(* Logix 5000 project; controller Amvex_Thorpe_Flowmeter vendor 1 type 14 code 106 rev 33.13; software revision 33.01; part 12 of 16 *)
(* tags used below, declared in another part *)
   Auto_Seq : SEQ;
   Barcode_Latch : BOOL;
   Barcode_Result_DATA : SINT[128];
   FAULTED : DINT;
   InfeedPalletTM1 : TIMER;
   Lift_stop_timer : TIMER;
   Manual_ONS : BOOL;
   MODE : MODE;
   Part_count : DINT;
   Test : Connect;
   Test_ONS : BOOL[32];
   Barcode_Data_String : STRING;
   Barcode_Delay : TIMER;
   Close : BOOL;
   Close_Rapid : Servo_Move;
   Close_Step : Servo_Move;
   Empty_Pallet_Timer : TIMER;
   Empty_Pallet_Timer2 : TIMER;
   Fastest_Delay : TIMER;
   In_Cycle : BOOL;
   Last_Test_Data : REAL[8];
   MCP : MCP;
   Open : BOOL;
   PH_Debug : DINT;
   Reject : BOOL;
   Reject_Barcode : BOOL;
   Reject_Pallet_Bit : DINT;
   Safety_OK : BOOL;
   Test2_Step : Servo_Move;
   Test3_Step : Servo_Move;
   Test4_Step : Servo_Move;
   Test5_Step : Servo_Move;
   Test_Data : REAL[8];
   Test_Data_Moved : BOOL;
   Test_Data_ONS : BOOL[32];
   Test_Delay_TMR : TIMER[5];
   Transmit_Data : BOOL;
   Vision_Result_OK_TMR : TIMER[6];
   Vision_TMR : TIMER[3];
(* MCP_Main, continued *)

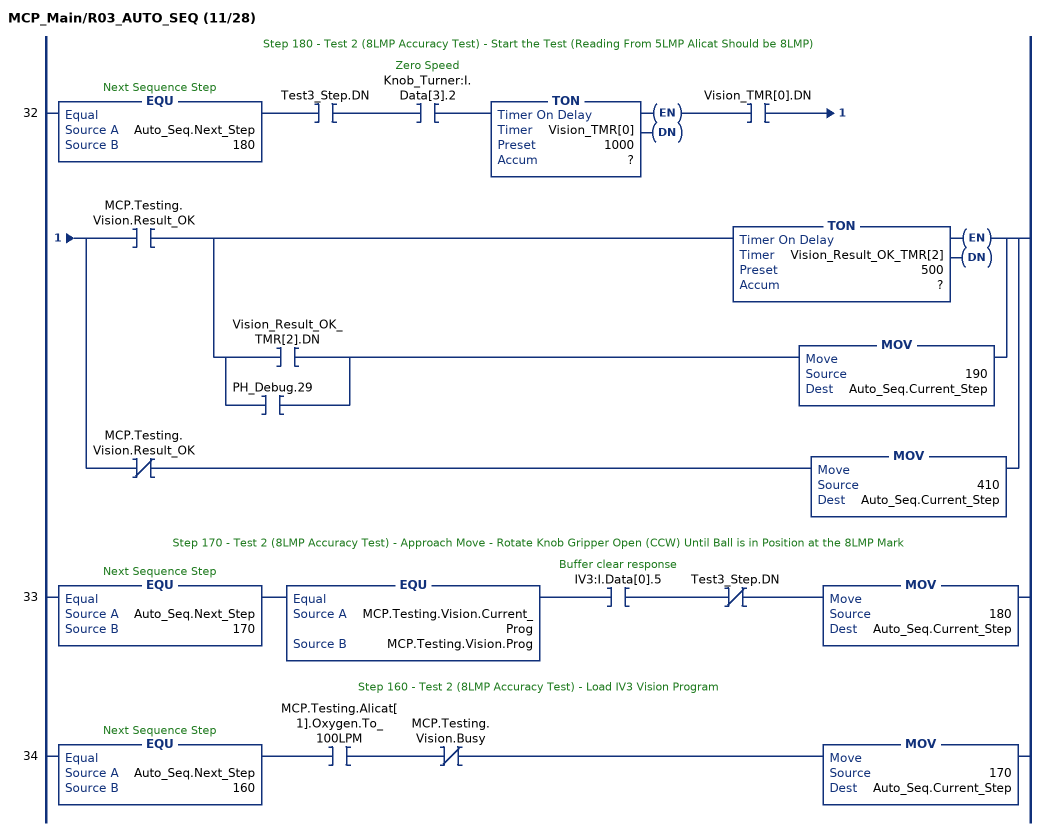
   [picture p212: MCP_Main/R03_AUTO_SEQ rungs 32-34]
   // Step 180 - Test 2 (8LMP Accuracy Test) - Start the Test (Reading From 5LMP Alicat Should be 8LMP)
   32: EQU(Auto_Seq.Next_Step,180)XIC(Test3_Step.DN)XIC(Knob_Turner:I.Data[3].2)TON(Vision_TMR[0],?,?)XIC(Vision_TMR[0].DN)[XIC(MCP.Testing.Vision.Result_OK) [TON(Vision_Result_OK_TMR[2],?,?) ,[XIC(Vision_Result_OK_TMR[2].DN) ,XIC(PH_Debug.29) ] MOV(190,Auto_Seq.Current_Step) ] ,XIO(MCP.Testing.Vision.Result_OK) MOV(410,Auto_Seq.Current_Step) ];
   // Step 170 - Test 2 (8LMP Accuracy Test) - Approach Move - Rotate Knob Gripper Open (CCW) Until Ball is in Position at the 8LMP Mark
   33: EQU(Auto_Seq.Next_Step,170)EQU(MCP.Testing.Vision.Current_Prog,MCP.Testing.Vision.Prog)XIC(IV3:I.Data[0].5)XIO(Test3_Step.DN)MOV(180,Auto_Seq.Current_Step);
   // Step 160 - Test 2 (8LMP Accuracy Test) - Load IV3 Vision Program
   34: EQU(Auto_Seq.Next_Step,160)XIC(MCP.Testing.Alicat[1].Oxygen.To_100LPM)XIO(MCP.Testing.Vision.Busy)MOV(170,Auto_Seq.Current_Step);
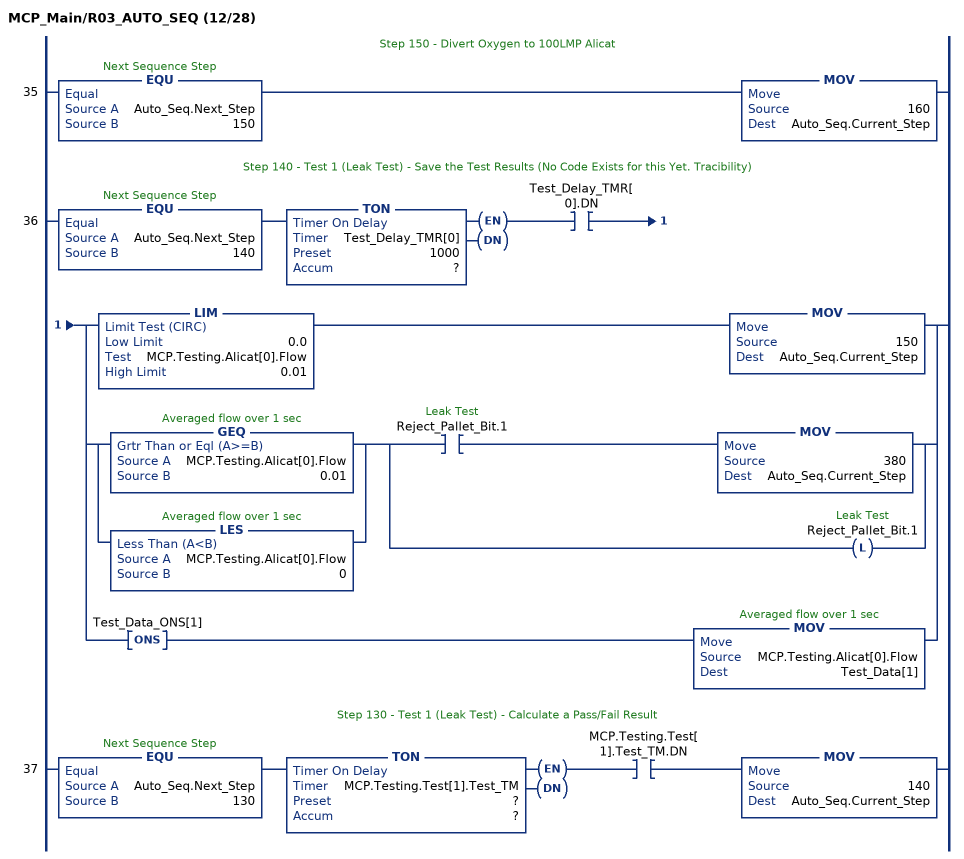
   // Step 150 - Divert Oxygen to 100LMP Alicat
   35: EQU(Auto_Seq.Next_Step,150)MOV(160,Auto_Seq.Current_Step);
   // Step 140 - Test 1 (Leak Test) - Save the Test Results (No Code Exists for this Yet. Tracibility)
   36: EQU(Auto_Seq.Next_Step,140)TON(Test_Delay_TMR[0],?,?)XIC(Test_Delay_TMR[0].DN)[LIM(0.0,MCP.Testing.Alicat[0].Flow,0.01) MOV(150,Auto_Seq.Current_Step) ,[GEQ(MCP.Testing.Alicat[0].Flow,0.01) ,LES(MCP.Testing.Alicat[0].Flow,0) ] [XIC(Reject_Pallet_Bit.1) MOV(380,Auto_Seq.Current_Step) ,OTL(Reject_Pallet_Bit.1) ] ,ONS(Test_Data_ONS[1]) MOV(MCP.Testing.Alicat[0].Flow,Test_Data[1]) ];
   // Step 130 - Test 1 (Leak Test) - Calculate a Pass/Fail Result
   37: EQU(Auto_Seq.Next_Step,130)TON(MCP.Testing.Test[1].Test_TM,?,?)XIC(MCP.Testing.Test[1].Test_TM.DN)MOV(140,Auto_Seq.Current_Step);
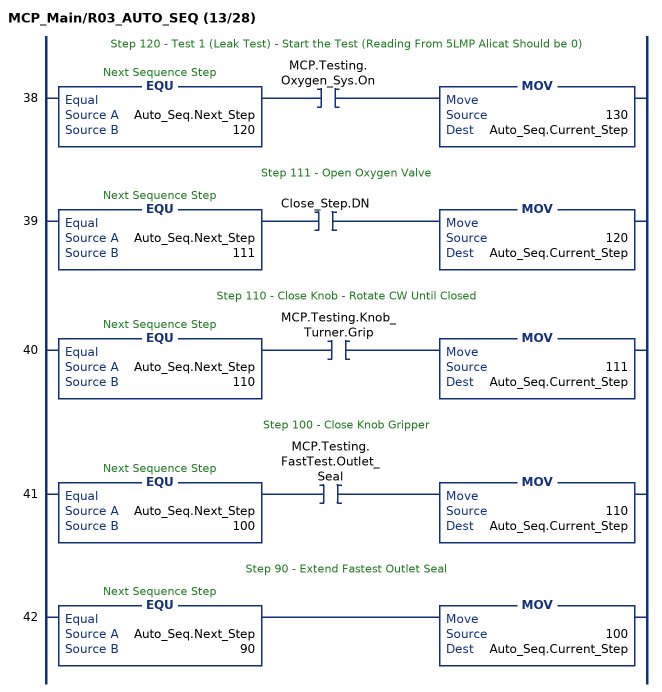
   // Step 120 - Test 1 (Leak Test) - Start the Test (Reading From 5LMP Alicat Should be 0)
   38: EQU(Auto_Seq.Next_Step,120)XIC(MCP.Testing.Oxygen_Sys.On)MOV(130,Auto_Seq.Current_Step);
   // Step 111 - Open Oxygen Valve
   39: EQU(Auto_Seq.Next_Step,111)XIC(Close_Step.DN)MOV(120,Auto_Seq.Current_Step);
   // Step 110 - Close Knob - Rotate CW Until Closed
   40: EQU(Auto_Seq.Next_Step,110)XIC(MCP.Testing.Knob_Turner.Grip)MOV(111,Auto_Seq.Current_Step);
   // Step 100 - Close Knob Gripper
   41: EQU(Auto_Seq.Next_Step,100)XIC(MCP.Testing.FastTest.Outlet_Seal)MOV(110,Auto_Seq.Current_Step);
   // Step 90 - Extend Fastest Outlet Seal
   42: EQU(Auto_Seq.Next_Step,90)MOV(100,Auto_Seq.Current_Step);
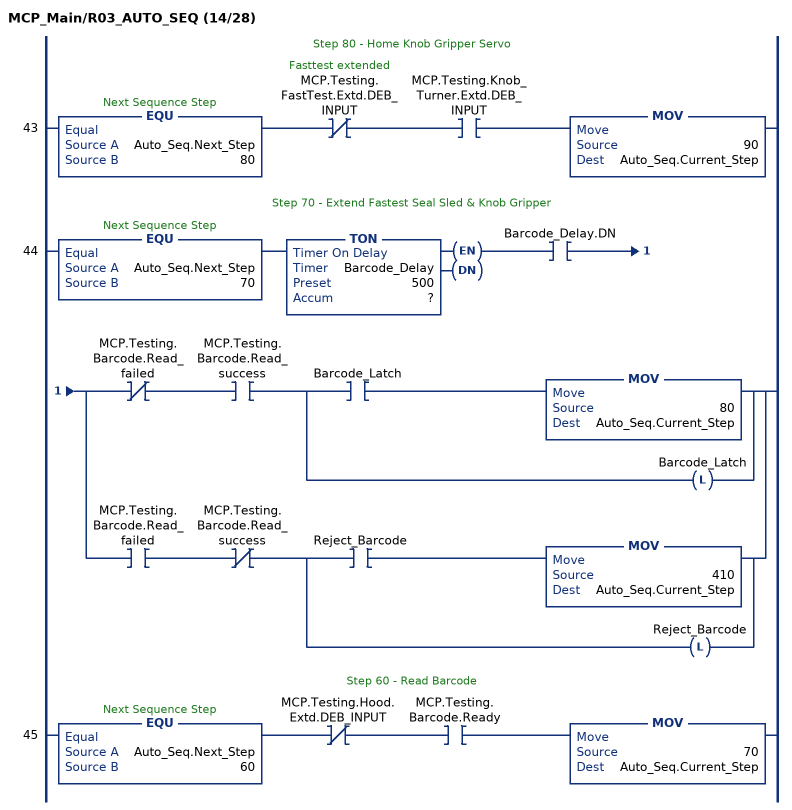
   // Step 80 - Home Knob Gripper Servo
   43: EQU(Auto_Seq.Next_Step,80)XIO(MCP.Testing.FastTest.Extd.DEB_INPUT)XIC(MCP.Testing.Knob_Turner.Extd.DEB_INPUT)MOV(90,Auto_Seq.Current_Step);
   // Step 70 - Extend Fastest Seal Sled & Knob Gripper
   44: EQU(Auto_Seq.Next_Step,70)TON(Barcode_Delay,?,?)XIC(Barcode_Delay.DN)[XIO(MCP.Testing.Barcode.Read_failed) XIC(MCP.Testing.Barcode.Read_success) [XIC(Barcode_Latch) MOV(80,Auto_Seq.Current_Step) ,OTL(Barcode_Latch) ] ,XIC(MCP.Testing.Barcode.Read_failed) XIO(MCP.Testing.Barcode.Read_success) [XIC(Reject_Barcode) MOV(410,Auto_Seq.Current_Step) ,OTL(Reject_Barcode) ] ];
   // Step 60 - Read Barcode
   45: EQU(Auto_Seq.Next_Step,60)XIO(MCP.Testing.Hood.Extd.DEB_INPUT)XIC(MCP.Testing.Barcode.Ready)MOV(70,Auto_Seq.Current_Step);
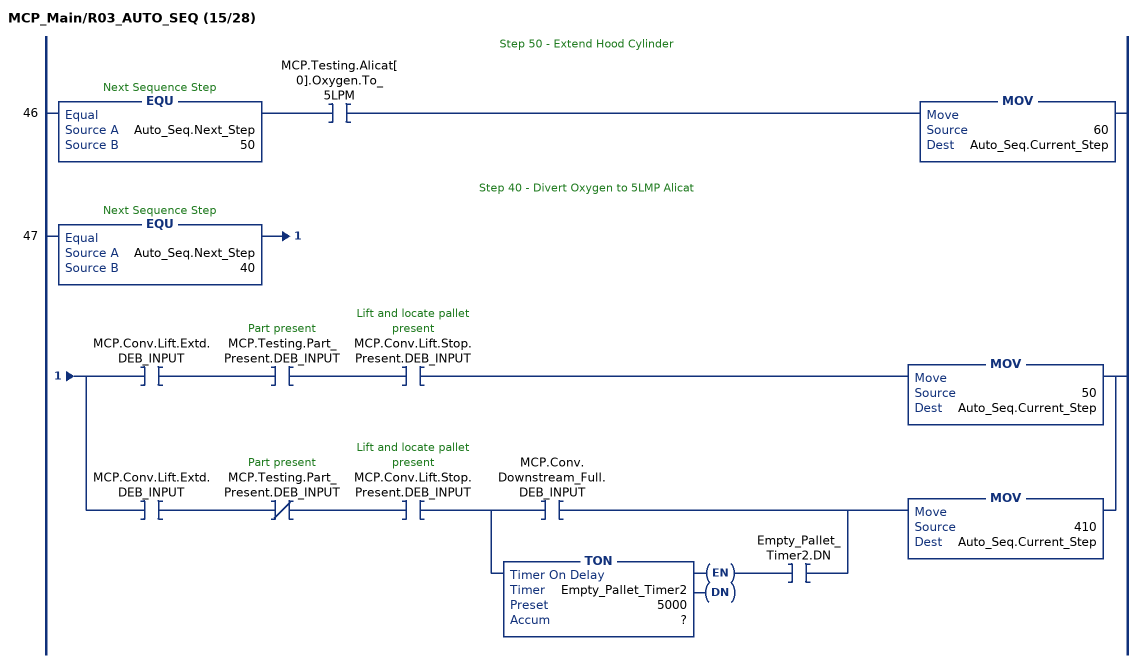
   // Step 50 - Extend Hood Cylinder
   46: EQU(Auto_Seq.Next_Step,50)XIC(MCP.Testing.Alicat[0].Oxygen.To_5LPM)MOV(60,Auto_Seq.Current_Step);
   // Step 40 - Divert Oxygen to 5LMP Alicat
   47: EQU(Auto_Seq.Next_Step,40)[XIC(MCP.Conv.Lift.Extd.DEB_INPUT) XIC(MCP.Testing.Part_Present.DEB_INPUT) XIC(MCP.Conv.Lift.Stop.Present.DEB_INPUT) MOV(50,Auto_Seq.Current_Step) ,XIC(MCP.Conv.Lift.Extd.DEB_INPUT) XIO(MCP.Testing.Part_Present.DEB_INPUT) XIC(MCP.Conv.Lift.Stop.Present.DEB_INPUT) [XIC(MCP.Conv.Downstream_Full.DEB_INPUT) ,TON(Empty_Pallet_Timer2,?,?) XIC(Empty_Pallet_Timer2.DN) ] MOV(410,Auto_Seq.Current_Step) ];
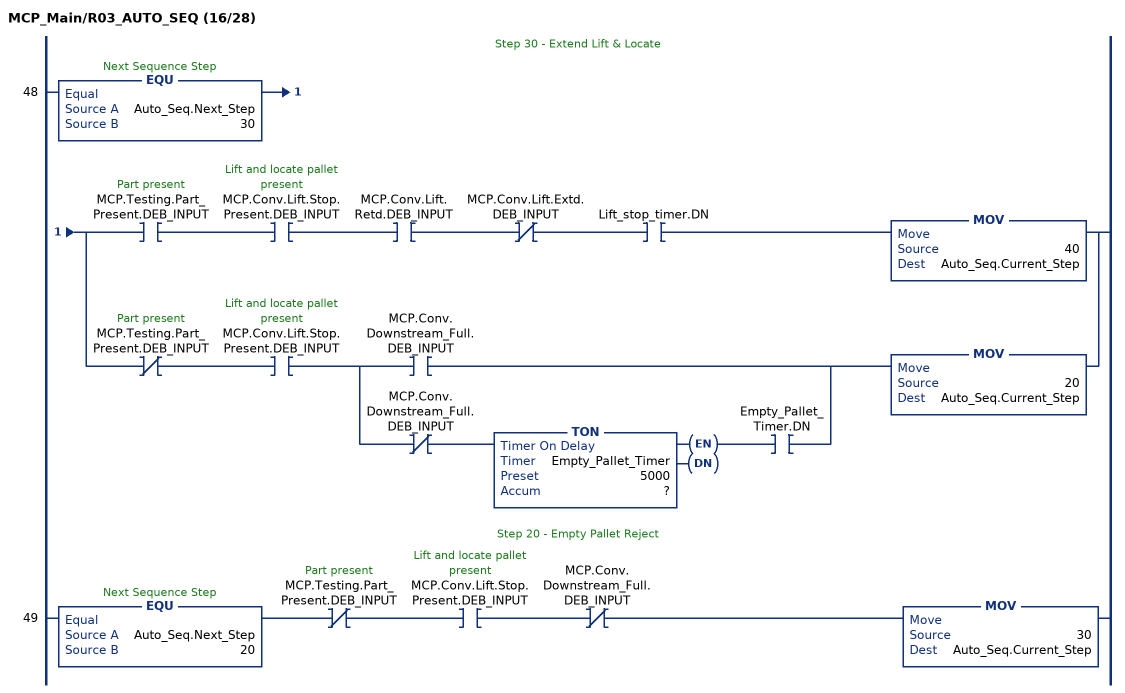
   // Step 30 - Extend Lift & Locate
   48: EQU(Auto_Seq.Next_Step,30)[XIC(MCP.Testing.Part_Present.DEB_INPUT) XIC(MCP.Conv.Lift.Stop.Present.DEB_INPUT) XIC(MCP.Conv.Lift.Retd.DEB_INPUT) XIO(MCP.Conv.Lift.Extd.DEB_INPUT) XIC(Lift_stop_timer.DN) MOV(40,Auto_Seq.Current_Step) ,XIO(MCP.Testing.Part_Present.DEB_INPUT) XIC(MCP.Conv.Lift.Stop.Present.DEB_INPUT) [XIC(MCP.Conv.Downstream_Full.DEB_INPUT) ,XIO(MCP.Conv.Downstream_Full.DEB_INPUT) TON(Empty_Pallet_Timer,?,?) XIC(Empty_Pallet_Timer.DN) ] MOV(20,Auto_Seq.Current_Step) ];
   // Step 20 - Empty Pallet Reject
   49: EQU(Auto_Seq.Next_Step,20)XIO(MCP.Testing.Part_Present.DEB_INPUT)XIC(MCP.Conv.Lift.Stop.Present.DEB_INPUT)XIO(MCP.Conv.Downstream_Full.DEB_INPUT)MOV(30,Auto_Seq.Current_Step);
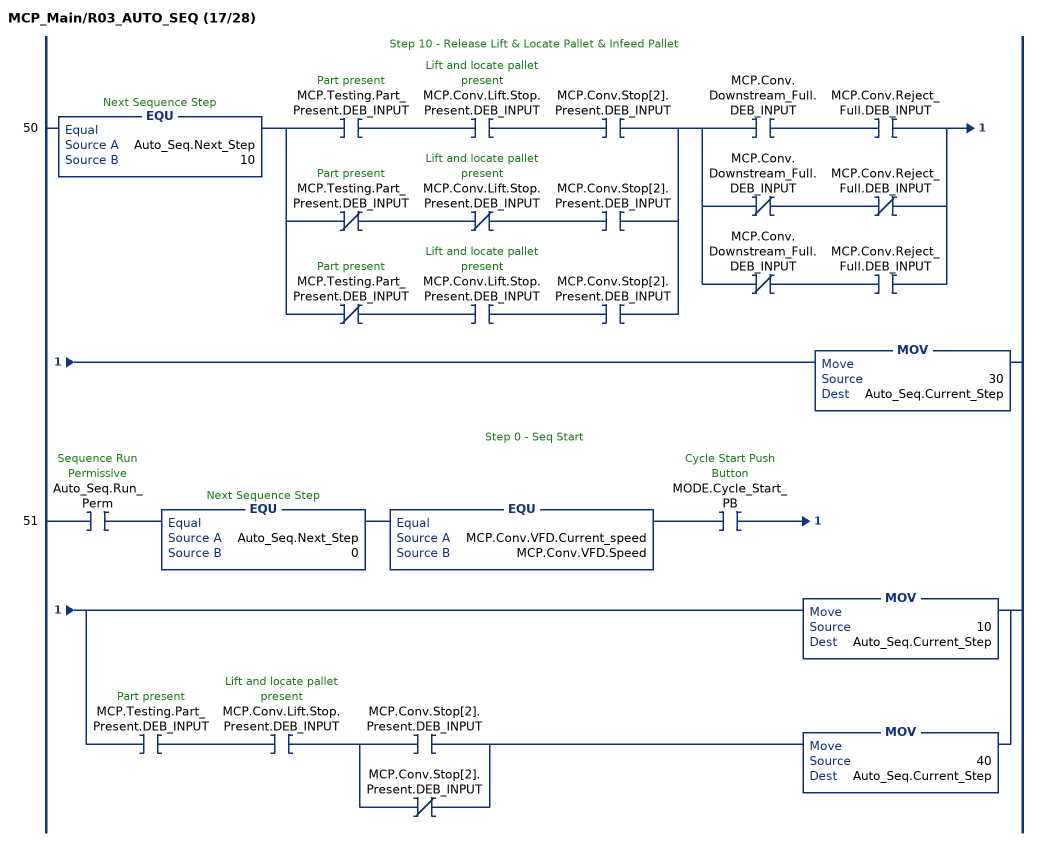
   // Step 10 - Release Lift & Locate Pallet & Infeed Pallet
   50: EQU(Auto_Seq.Next_Step,10)[XIC(MCP.Testing.Part_Present.DEB_INPUT) XIC(MCP.Conv.Lift.Stop.Present.DEB_INPUT) XIC(MCP.Conv.Stop[2].Present.DEB_INPUT) ,XIO(MCP.Testing.Part_Present.DEB_INPUT) XIO(MCP.Conv.Lift.Stop.Present.DEB_INPUT) XIC(MCP.Conv.Stop[2].Present.DEB_INPUT) ,XIO(MCP.Testing.Part_Present.DEB_INPUT) XIC(MCP.Conv.Lift.Stop.Present.DEB_INPUT) XIC(MCP.Conv.Stop[2].Present.DEB_INPUT) ][XIC(MCP.Conv.Downstream_Full.DEB_INPUT) XIC(MCP.Conv.Reject_Full.DEB_INPUT) ,XIO(MCP.Conv.Downstream_Full.DEB_INPUT) XIO(MCP.Conv.Reject_Full.DEB_INPUT) ,XIO(MCP.Conv.Downstream_Full.DEB_INPUT) XIC(MCP.Conv.Reject_Full.DEB_INPUT) ]MOV(30,Auto_Seq.Current_Step);
   // Step 0 - Seq Start
   51: XIC(Auto_Seq.Run_Perm)EQU(Auto_Seq.Next_Step,0)EQU(MCP.Conv.VFD.Current_speed,MCP.Conv.VFD.Speed)XIC(MODE.Cycle_Start_PB)[MOV(10,Auto_Seq.Current_Step) ,XIC(MCP.Testing.Part_Present.DEB_INPUT) XIC(MCP.Conv.Lift.Stop.Present.DEB_INPUT) [XIC(MCP.Conv.Stop[2].Present.DEB_INPUT) ,XIO(MCP.Conv.Stop[2].Present.DEB_INPUT) ] MOV(40,Auto_Seq.Current_Step) ];
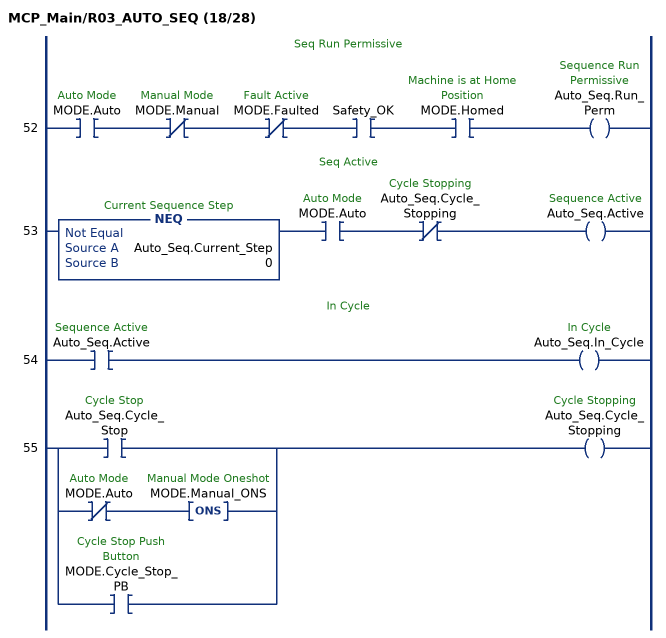
   // Seq Run Permissive
   52: XIC(MODE.Auto)XIO(MODE.Manual)XIO(MODE.Faulted)XIC(Safety_OK)XIC(MODE.Homed)OTE(Auto_Seq.Run_Perm);
   // Seq Active
   53: NEQ(Auto_Seq.Current_Step,0)XIC(MODE.Auto)XIO(Auto_Seq.Cycle_Stopping)OTE(Auto_Seq.Active);
   // In Cycle
   54: XIC(Auto_Seq.Active)OTE(Auto_Seq.In_Cycle);
   55: [XIC(Auto_Seq.Cycle_Stop) ,XIO(MODE.Auto) ONS(MODE.Manual_ONS) ,XIC(MODE.Cycle_Stop_PB) ]OTE(Auto_Seq.Cycle_Stopping);
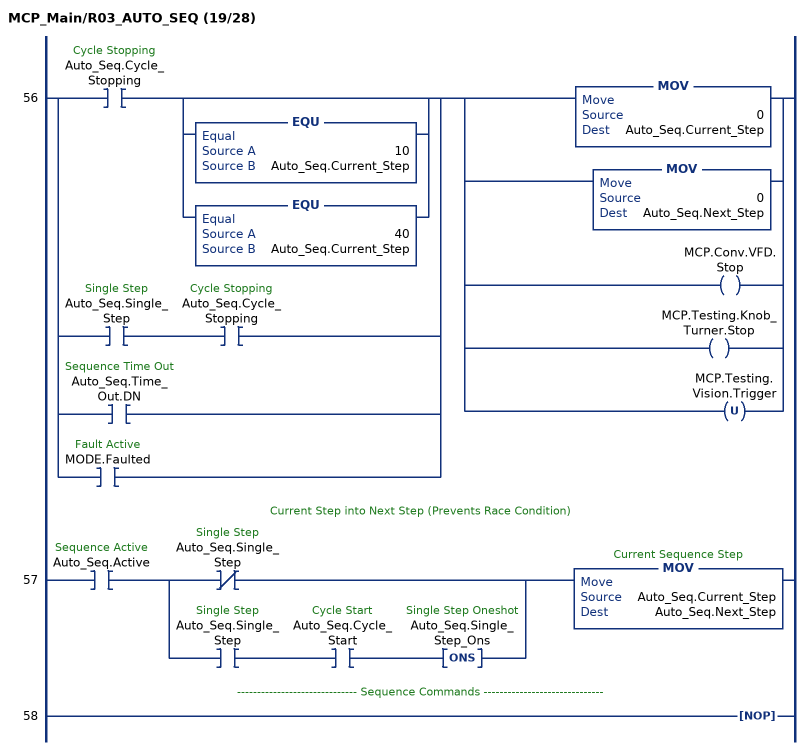
   56: [XIC(Auto_Seq.Cycle_Stopping) [,EQU(10,Auto_Seq.Current_Step) ,EQU(40,Auto_Seq.Current_Step) ] ,XIC(Auto_Seq.Single_Step) XIC(Auto_Seq.Cycle_Stopping) ,XIC(Auto_Seq.Time_Out.DN) ,XIC(MODE.Faulted) ][MOV(0,Auto_Seq.Current_Step) ,MOV(0,Auto_Seq.Next_Step) ,OTE(MCP.Conv.VFD.Stop) ,OTE(MCP.Testing.Knob_Turner.Stop) ,OTU(MCP.Testing.Vision.Trigger) ];
   // Current Step into Next Step (Prevents Race Condition)
   57: XIC(Auto_Seq.Active)[XIO(Auto_Seq.Single_Step) ,XIC(Auto_Seq.Single_Step) XIC(Auto_Seq.Cycle_Start) ONS(Auto_Seq.Single_Step_Ons) ]MOV(Auto_Seq.Current_Step,Auto_Seq.Next_Step);
   // ------------------------------ Sequence Commands ------------------------------
   58: NOP();
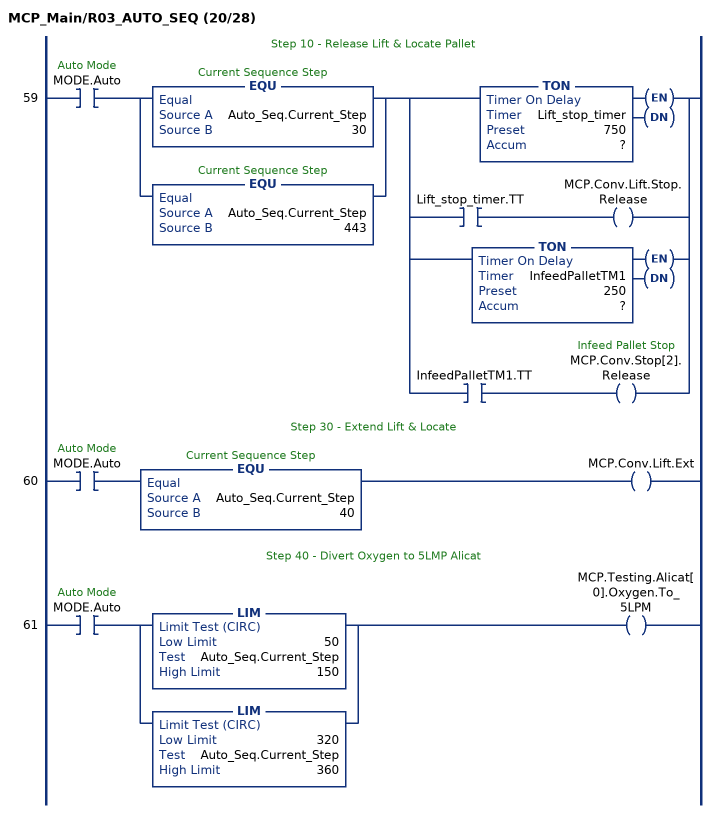
   // Step 10 - Release Lift & Locate Pallet
   59: XIC(MODE.Auto)[EQU(Auto_Seq.Current_Step,30) ,EQU(Auto_Seq.Current_Step,443) ][[TON(Lift_stop_timer,?,?) ,XIC(Lift_stop_timer.TT) OTE(MCP.Conv.Lift.Stop.Release) ] ,[TON(InfeedPalletTM1,?,?) ,XIC(InfeedPalletTM1.TT) OTE(MCP.Conv.Stop[2].Release) ] ];
   // Step 30 - Extend Lift & Locate
   60: XIC(MODE.Auto)EQU(Auto_Seq.Current_Step,40)OTE(MCP.Conv.Lift.Ext);
   // Step 40 - Divert Oxygen to 5LMP Alicat
   61: XIC(MODE.Auto)[LIM(50,Auto_Seq.Current_Step,150) ,LIM(320,Auto_Seq.Current_Step,360) ]OTE(MCP.Testing.Alicat[0].Oxygen.To_5LPM);
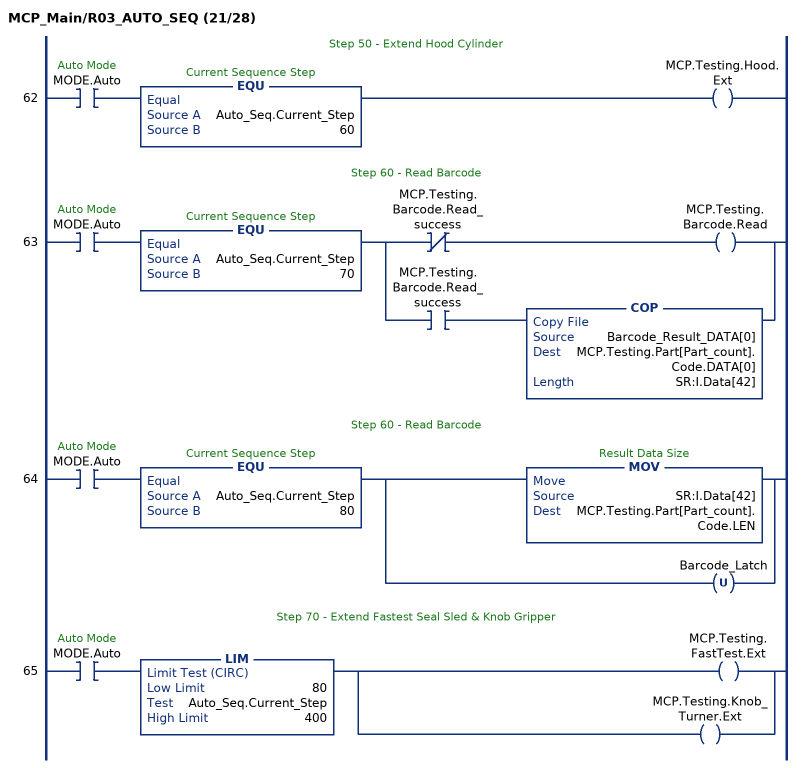
   // Step 50 - Extend Hood Cylinder
   62: XIC(MODE.Auto)EQU(Auto_Seq.Current_Step,60)OTE(MCP.Testing.Hood.Ext);
   // Step 60 - Read Barcode
   63: XIC(MODE.Auto)EQU(Auto_Seq.Current_Step,70)[XIO(MCP.Testing.Barcode.Read_success) OTE(MCP.Testing.Barcode.Read) ,XIC(MCP.Testing.Barcode.Read_success) COP(Barcode_Result_DATA[0],MCP.Testing.Part[Part_count].Code.DATA[0],SR:I.Data[42]) ];
   // Step 60 - Read Barcode
   64: XIC(MODE.Auto)EQU(Auto_Seq.Current_Step,80)[MOV(SR:I.Data[42],MCP.Testing.Part[Part_count].Code.LEN) ,OTU(Barcode_Latch) ];
   // Step 70 - Extend Fastest Seal Sled & Knob Gripper
   65: XIC(MODE.Auto)LIM(80,Auto_Seq.Current_Step,400)[OTE(MCP.Testing.FastTest.Ext) ,OTE(MCP.Testing.Knob_Turner.Ext) ];
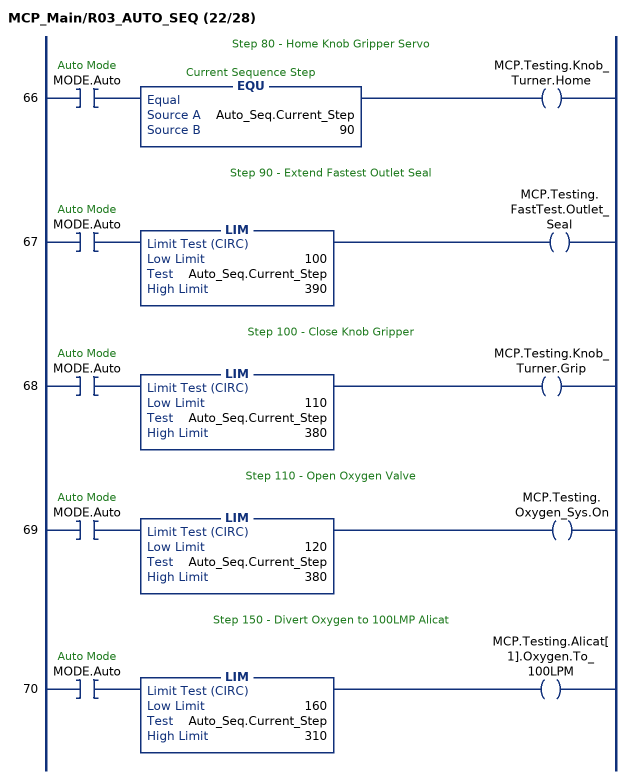
   // Step 80 - Home Knob Gripper Servo
   66: XIC(MODE.Auto)EQU(Auto_Seq.Current_Step,90)OTE(MCP.Testing.Knob_Turner.Home);
   // Step 90 - Extend Fastest Outlet Seal
   67: XIC(MODE.Auto)LIM(100,Auto_Seq.Current_Step,390)OTE(MCP.Testing.FastTest.Outlet_Seal);
   // Step 100 - Close Knob Gripper
   68: XIC(MODE.Auto)LIM(110,Auto_Seq.Current_Step,380)OTE(MCP.Testing.Knob_Turner.Grip);
   // Step 110 - Open Oxygen Valve
   69: XIC(MODE.Auto)LIM(120,Auto_Seq.Current_Step,380)OTE(MCP.Testing.Oxygen_Sys.On);
   // Step 150 - Divert Oxygen to 100LMP Alicat
   70: XIC(MODE.Auto)LIM(160,Auto_Seq.Current_Step,310)OTE(MCP.Testing.Alicat[1].Oxygen.To_100LPM);
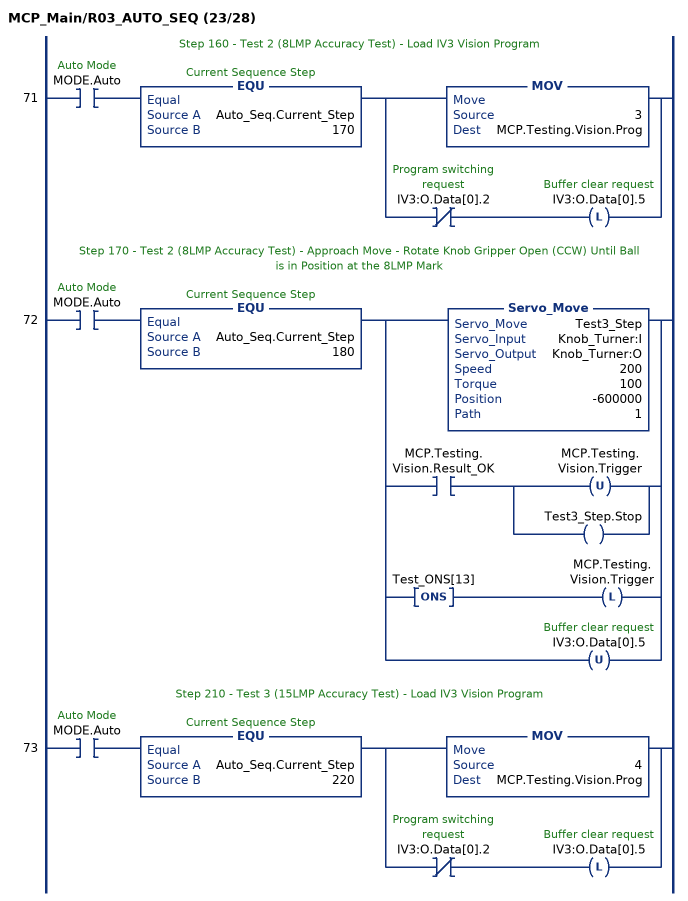
   // Step 160 - Test 2 (8LMP Accuracy Test) - Load IV3 Vision Program
   71: XIC(MODE.Auto)EQU(Auto_Seq.Current_Step,170)[MOV(3,MCP.Testing.Vision.Prog) ,XIO(IV3:O.Data[0].2) OTL(IV3:O.Data[0].5) ];
   // Step 170 - Test 2 (8LMP Accuracy Test) - Approach Move - Rotate Knob Gripper Open (CCW) Until Ball is in Position at the 8LMP Mark
   72: XIC(MODE.Auto)EQU(Auto_Seq.Current_Step,180)[Servo_Move(Test3_Step,Knob_Turner:I,Knob_Turner:O,200,100,-600000,1) ,XIC(MCP.Testing.Vision.Result_OK) [OTU(MCP.Testing.Vision.Trigger) ,OTE(Test3_Step.Stop) ] ,ONS(Test_ONS[13]) OTL(MCP.Testing.Vision.Trigger) ,OTU(IV3:O.Data[0].5) ];
   // Step 210 - Test 3 (15LMP Accuracy Test) - Load IV3 Vision Program
   73: XIC(MODE.Auto)EQU(Auto_Seq.Current_Step,220)[MOV(4,MCP.Testing.Vision.Prog) ,XIO(IV3:O.Data[0].2) OTL(IV3:O.Data[0].5) ];
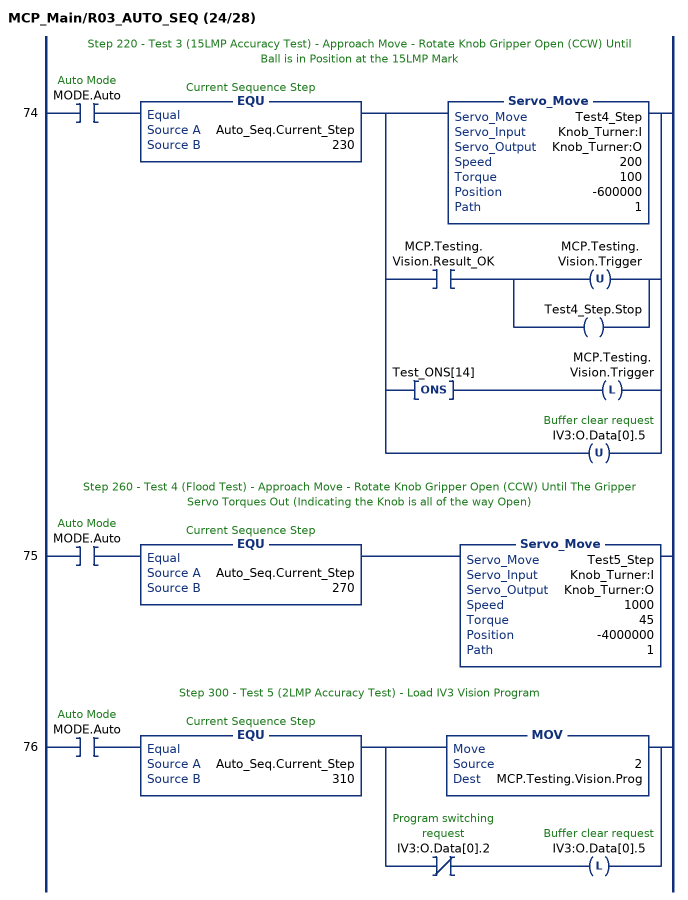
   // Step 220 - Test 3 (15LMP Accuracy Test) - Approach Move - Rotate Knob Gripper Open (CCW) Until Ball is in Position at the 15LMP Mark
   74: XIC(MODE.Auto)EQU(Auto_Seq.Current_Step,230)[Servo_Move(Test4_Step,Knob_Turner:I,Knob_Turner:O,200,100,-600000,1) ,XIC(MCP.Testing.Vision.Result_OK) [OTU(MCP.Testing.Vision.Trigger) ,OTE(Test4_Step.Stop) ] ,ONS(Test_ONS[14]) OTL(MCP.Testing.Vision.Trigger) ,OTU(IV3:O.Data[0].5) ];
   // Step 260 - Test 4 (Flood Test) - Approach Move - Rotate Knob Gripper Open (CCW) Until The Gripper Servo Torques Out (Indicating the Knob is all of the way Open)
   75: XIC(MODE.Auto)EQU(Auto_Seq.Current_Step,270)Servo_Move(Test5_Step,Knob_Turner:I,Knob_Turner:O,1000,45,-4000000,1);
   // Step 300 - Test 5 (2LMP Accuracy Test) - Load IV3 Vision Program
   76: XIC(MODE.Auto)EQU(Auto_Seq.Current_Step,310)[MOV(2,MCP.Testing.Vision.Prog) ,XIO(IV3:O.Data[0].2) OTL(IV3:O.Data[0].5) ];
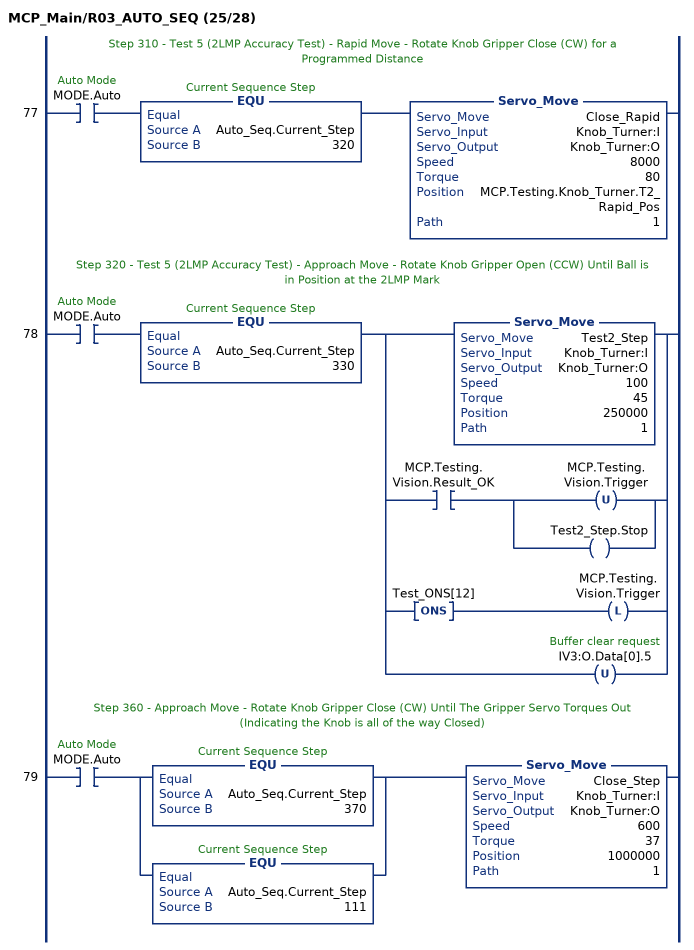
   // Step 310 - Test 5 (2LMP Accuracy Test) - Rapid Move - Rotate Knob Gripper Close (CW) for a Programmed Distance
   77: XIC(MODE.Auto)EQU(Auto_Seq.Current_Step,320)Servo_Move(Close_Rapid,Knob_Turner:I,Knob_Turner:O,8000,80,MCP.Testing.Knob_Turner.T2_Rapid_Pos,1);
   // Step 320 - Test 5 (2LMP Accuracy Test) - Approach Move - Rotate Knob Gripper Open (CCW) Until Ball is in Position at the 2LMP Mark
   78: XIC(MODE.Auto)EQU(Auto_Seq.Current_Step,330)[Servo_Move(Test2_Step,Knob_Turner:I,Knob_Turner:O,100,45,250000,1) ,XIC(MCP.Testing.Vision.Result_OK) [OTU(MCP.Testing.Vision.Trigger) ,OTE(Test2_Step.Stop) ] ,ONS(Test_ONS[12]) OTL(MCP.Testing.Vision.Trigger) ,OTU(IV3:O.Data[0].5) ];
   // Step 360 - Approach Move - Rotate Knob Gripper Close (CW) Until The Gripper Servo Torques Out (Indicating the Knob is all of the way Closed)
   79: XIC(MODE.Auto)[EQU(Auto_Seq.Current_Step,370) ,EQU(Auto_Seq.Current_Step,111) ]Servo_Move(Close_Step,Knob_Turner:I,Knob_Turner:O,600,37,1000000,1);
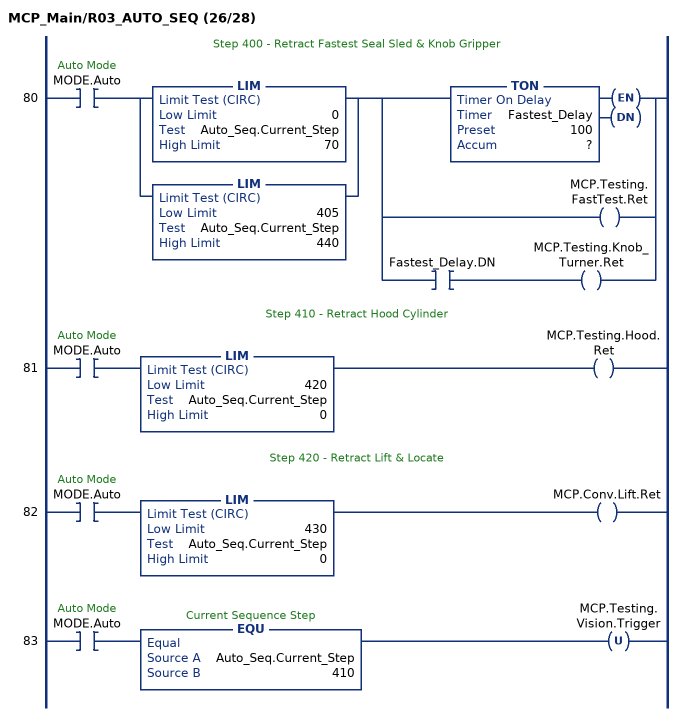
   // Step 400 - Retract Fastest Seal Sled & Knob Gripper
   80: XIC(MODE.Auto)[LIM(0,Auto_Seq.Current_Step,70) ,LIM(405,Auto_Seq.Current_Step,440) ][TON(Fastest_Delay,?,?) ,OTE(MCP.Testing.FastTest.Ret) ,XIC(Fastest_Delay.DN) OTE(MCP.Testing.Knob_Turner.Ret) ];
   // Step 410 - Retract Hood Cylinder
   81: XIC(MODE.Auto)LIM(420,Auto_Seq.Current_Step,0)OTE(MCP.Testing.Hood.Ret);
   // Step 420 - Retract Lift & Locate
   82: XIC(MODE.Auto)LIM(430,Auto_Seq.Current_Step,0)OTE(MCP.Conv.Lift.Ret);
   83: XIC(MODE.Auto)EQU(Auto_Seq.Current_Step,410)OTU(MCP.Testing.Vision.Trigger);
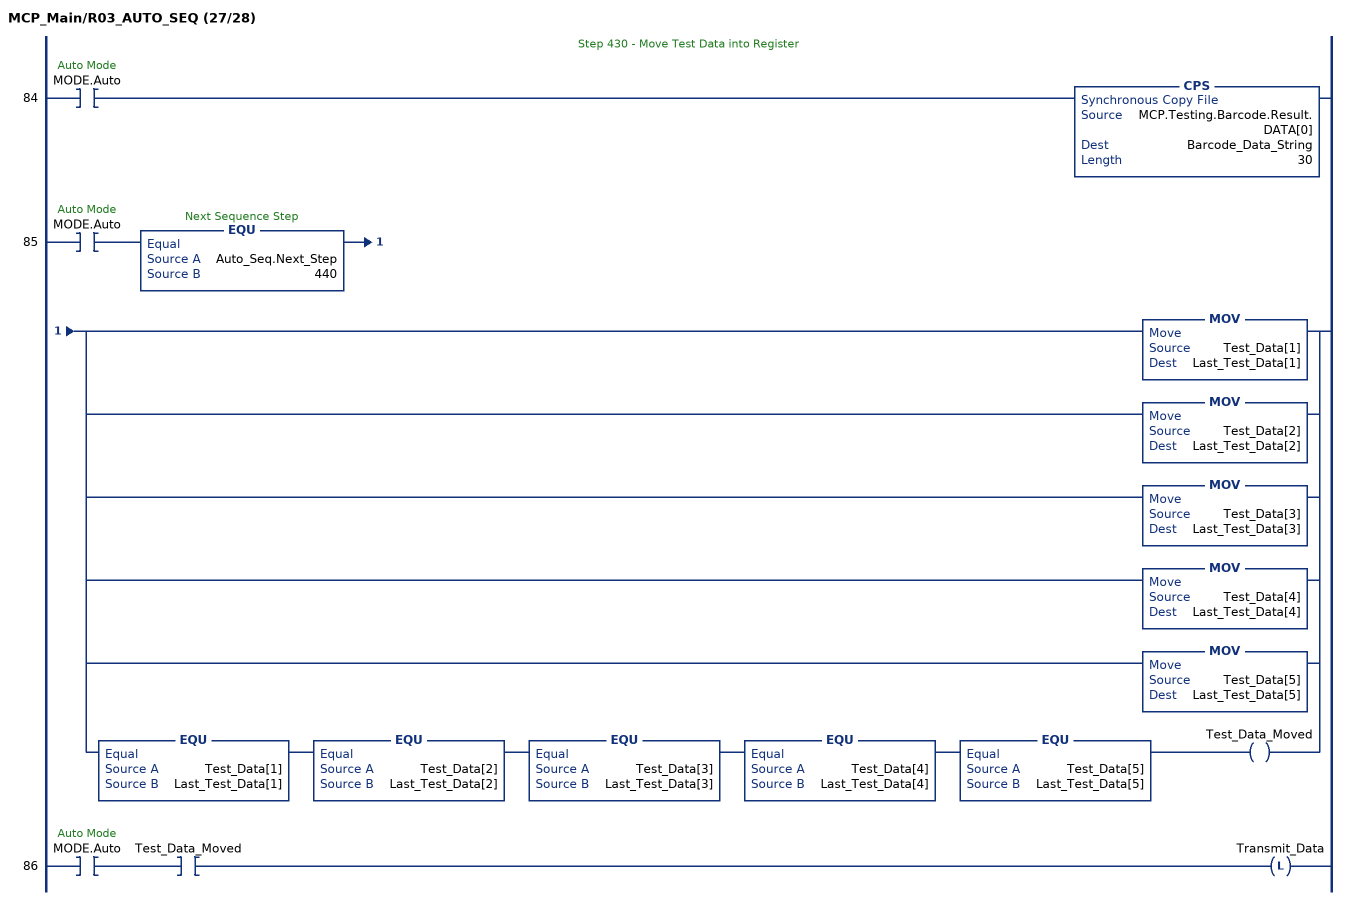
   // Step 430 - Move Test Data into Register
   84: XIC(MODE.Auto)CPS(MCP.Testing.Barcode.Result.DATA[0],Barcode_Data_String,30);
   85: XIC(MODE.Auto)EQU(Auto_Seq.Next_Step,440)[MOV(Test_Data[1],Last_Test_Data[1]) ,MOV(Test_Data[2],Last_Test_Data[2]) ,MOV(Test_Data[3],Last_Test_Data[3]) ,MOV(Test_Data[4],Last_Test_Data[4]) ,MOV(Test_Data[5],Last_Test_Data[5]) ,EQU(Test_Data[1],Last_Test_Data[1]) EQU(Test_Data[2],Last_Test_Data[2]) EQU(Test_Data[3],Last_Test_Data[3]) EQU(Test_Data[4],Last_Test_Data[4]) EQU(Test_Data[5],Last_Test_Data[5]) OTE(Test_Data_Moved) ];
   86: XIC(MODE.Auto)XIC(Test_Data_Moved)OTL(Transmit_Data);
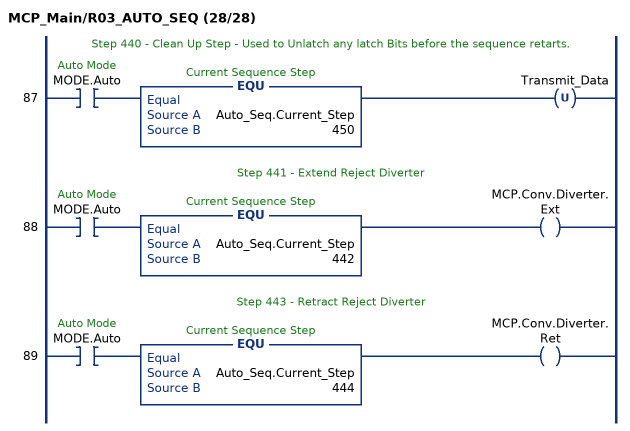
   // Step 440 - Clean Up Step - Used to Unlatch any latch Bits before the sequence retarts.
   87: XIC(MODE.Auto)EQU(Auto_Seq.Current_Step,450)OTU(Transmit_Data);
   // Step 441 - Extend Reject Diverter
   88: XIC(MODE.Auto)EQU(Auto_Seq.Current_Step,442)OTE(MCP.Conv.Diverter.Ext);
   // Step 443 - Retract Reject Diverter
   89: XIC(MODE.Auto)EQU(Auto_Seq.Current_Step,444)OTE(MCP.Conv.Diverter.Ret);
END_ROUTINE
